FUNCTION_BLOCK AR_CALIBRATE (* Adapter-based two-point calibration (offset & scale) of an analog input *)
  (* Standard: 61499-1 *)
  (* Version 2.0, 2026-06-01, Meisterschulen am Ostbahnhof *)
  PACKAGE adapter::Engineering::measurements;
  (* Documentation:
  Formula
   Y = (X + OFFSET) * SCALE Calibration (Two-Point)
    - Offset (CO): Apply low reference, set Y_Offset to desired output, trigger CO
   OFFSET := Y_Offset - X → shifts X so that Y = Y_Offset * SCALE at this point
   Note: Only correct when SCALE = 1.
   - Scale (CS): Apply high reference, set Y_Scale to desired output, trigger CS
   SCALE := Y_Scale / (X + OFFSET) → scales so that Y = Y_Scale at this point
    Note: Both Y_Offset and Y_Scale are target values on the output side.
   ⚠ Order requirement: CO must be executed before CS, because CS uses OFFSET.
  *)
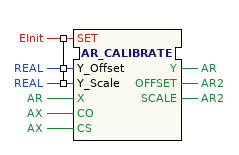
  EVENT_INPUT
    SET : EInit WITH Y_Offset, Y_Scale; (* Set References *)
  END_EVENT
  VAR_INPUT
    Y_Offset : REAL; (* Reference for offset calibration *)
    Y_Scale : REAL; (* Reference for scale calibration *)
  END_VAR
  SOCKETS
    X : adapter::types::unidirectional::AR; (* Input *)
    CO : adapter::types::unidirectional::AX; (* Calibrate Offset *)
    CS : adapter::types::unidirectional::AX; (* Calibrate Scale *)
  END_SOCKETS
  PLUGS
    Y : adapter::types::unidirectional::AR; (* Calibrated Output *)
    OFFSET : adapter::types::bidirectional::AR2; (* Offset value *)
    SCALE : adapter::types::bidirectional::AR2; (* Scale value *)
  END_PLUGS
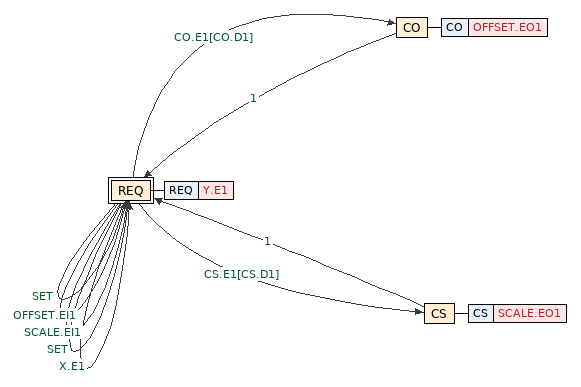
  EC_STATES
    REQ : REQ -> Y.E1;
    CO : CO -> OFFSET.EO1;
    CS : CS -> SCALE.EO1;
  END_STATES
  EC_TRANSITIONS
    REQ TO REQ := X.E1;
    REQ TO REQ := SET;
    REQ TO REQ := SET;
    REQ TO REQ := OFFSET.EI1;
    REQ TO REQ := SCALE.EI1;
    CO TO REQ := 1;
    CS TO REQ := 1;
    REQ TO CO := CO.E1[CO.D1];
    REQ TO CS := CS.E1[CS.D1];
  END_TRANSITIONS
  ALGORITHM REQ IN ST: (* REQ *)
(* calculate calibrated output *)
Y.D1 := (X.D1 + OFFSET.DI1) * SCALE.DI1;
  END_ALGORITHM
  ALGORITHM CO IN ST: (* CO *)
(* store offset so that Y = Y_Offset at current X *)
(* note: after CO, Y = Y_Offset * SCALE, only correct when SCALE = 1 *)
OFFSET.DO1 := Y_Offset - X.D1;
  END_ALGORITHM
  ALGORITHM CS IN ST: (* CS *)
(* store scale so that Y = Y_Scale at current X (requires OFFSET from CO!) *)
IF (X.D1 + OFFSET.DI1) <> 0.0 THEN
	SCALE.DO1 := Y_Scale / (X.D1 + OFFSET.DI1);
END_IF;
  END_ALGORITHM
END_FUNCTION_BLOCK
